FUNCTION_BLOCK itfStatusFlagsImplement IMPLEMENTS itfStatusFlags
VAR_INPUT
END_VAR
VAR_OUTPUT
END_VAR
VAR
	Buffering : BOOL;
	Dosing : BOOL;
	Fault : BOOL;
	HaltBatch : BOOL;
	Mixing : BOOL;
	Storing : BOOL;
	LowProduct : BOOL;
END_VAR

{warning 'add property implementation'}
PROPERTY pBuffering : BOOL
GET
pBuffering := Buffering;
END_GET
SET
Buffering := pBuffering;
END_SET
END_PROPERTY

{warning 'add property implementation'}
PROPERTY pDosing : BOOL
GET
pDosing := Dosing;
END_GET
SET
Dosing := pDosing;
END_SET
END_PROPERTY

{warning 'add property implementation'}
PROPERTY pFault : BOOL
GET
pFault := Fault;
END_GET
SET
Fault := pFault;
END_SET
END_PROPERTY

{warning 'add property implementation'}
PROPERTY pHaltBatch : BOOL
GET
pHaltBatch := HaltBatch;
END_GET
SET
HaltBatch := pHaltBatch;
END_SET
END_PROPERTY

{warning 'add property implementation'}
PROPERTY pLowProduct : BOOL
GET
pLowProduct := LowProduct;
END_GET
SET
LowProduct := pLowProduct;
END_SET
END_PROPERTY

{warning 'add property implementation'}
PROPERTY pMixing : BOOL
GET
pMixing := Mixing;
END_GET
SET
Mixing := pMixing;
END_SET
END_PROPERTY

{warning 'add property implementation'}
PROPERTY pStoring : BOOL
GET
pStoring := Storing;
END_GET
SET
Storing := pStoring;
END_SET
END_PROPERTY

END_FUNCTION_BLOCK

(* stored: Version 1.1.0.1, ProductVersion 3.1.4024.12
   POU itfStatusFlagsImplement: Id {b4afa069-e6e8-4aac-9778-c5758541973e}, SpecialFunc None
   Property pBuffering: Id {6ef13a59-15c8-415f-a35e-1c2f9592531a}
   Get Get: Id {9e5e72d9-d24c-45f8-9945-8bf0c0360e61}
   Set Set: Id {fef71d4d-2123-4605-b8e8-786f3ee8ca04}
   Property pDosing: Id {f5c379a8-e972-4625-aab4-371a51893e76}
   Get Get: Id {a1bc8ab2-e837-4b9f-954a-b22bacee030d}
   Set Set: Id {9d3b5002-40fc-4202-bfb2-8f20995ff8b1}
   Property pFault: Id {c99e1cf4-ad15-4a82-a27e-87ea2b59b061}
   Get Get: Id {70134aeb-5305-48ee-af8e-e485f2eb4f53}
   Set Set: Id {008214f4-1307-4532-a4af-45b13005caa8}
   Property pHaltBatch: Id {7e020721-f19f-46d5-8731-ff3a64d1b57e}
   Get Get: Id {c34c1fae-6c2f-4567-920c-9693936463d8}
   Set Set: Id {655a4ea4-fb05-41d0-836f-ee044658321a}
   Property pLowProduct: Id {9bb1f0e4-640f-4829-b516-d76094ad5eb3}
   Get Get: Id {c8648b14-02c6-45ca-9425-ce0772b3c90f}
   Set Set: Id {5c689d97-ddb5-464a-a69c-338a054533c4}
   Property pMixing: Id {8fde8687-0c07-4a21-9b35-9462bbde35a1}
   Get Get: Id {d015fff5-e404-441c-9e04-b6142a66232f}
   Set Set: Id {6d3ecc67-0300-408c-9ec4-126edff54f97}
   Property pStoring: Id {4d77a9a7-f347-4ac4-a52c-94a95f954e73}
   Get Get: Id {282f82d1-4822-4d99-b873-b68fb6c1f444}
   Set Set: Id {3803e5a8-5dfb-4b17-beb3-e18c30b1e95d} *)
